Yaskawa INFORM job: mini.JBI

/JOB
//NAME mini
//POS
///NPOS 0,0,0,0,0,0
///TOOL 1
///POSTYPE ROBOT
///RECTAN
///RCONF 1,0,0,0,0,0,0,0,0,0,0,0,0,0,0,0,0,0,0,0,0,0,0,0
//INST
///DATE 2021/02/10 13:51
///COMM
///ATTR SC,RW,RJ
////FRAME USER 2
///GROUP1 RB1
NOP
CALL JOB:DEBUT
'Part trajectory number: 0
CALL JOB:miniTRJ0
'Part trajectory number: 1
CALL JOB:miniTRJ1
'Part trajectory number: 2
CALL JOB:miniTRJ2
CALL JOB:FIN
END
